FUNCTION F_LeakMonitor_LIR_1 : FB_LeakMonitor
VAR_INPUT
END_VAR
VAR_OUTPUT
	// Provide stBoundaries output so test functions can reuse the boundaries
	stBoundaries : ST_LeakBoundaries := F_LeakBoundaries();
END_VAR
VAR
	fbLeakMonitor : FB_LeakMonitor;
END_VAR

fbLeakMonitor(
	bLeakDetected := TRUE,
	nLocationResistance := stBoundaries.nLMax6 - 1,
	stBound := stBoundaries
);

F_LeakMonitor_LIR_1 := fbLeakMonitor;

END_FUNCTION

(* stored: Version 1.1.0.1, ProductVersion 3.1.4024.0
   POU F_LeakMonitor_LIR_1: Id {e9d27db8-49ac-49da-b9ae-ffec0b53c69f}, SpecialFunc None *)
